PROGRAM PRG_ControlHMIInit
VAR
	(*	Konfiguracja HMIManager		*)
	fbDedaultHMIConfiguration		: FB_DefaultHMIConfiguration;
	fbHMIConfigure					: FB_HMIConfigure;
	
END_VAR

IF (NOT GVL_SystemVariable.bControlHMIInit) THEN
	GVL_SystemVariable.bControlHMIInit := TRUE;
		(*	Konfiguracjia systemu HMI	*)
	fbHMIConfigure.AddConfiguration (fbConfigure := fbDedaultHMIConfiguration);
	PRG_ControlHMI.fbHMIManager.AddModulConfigure (fbHMIConfigure := fbHMIConfigure);
	
END_IF

END_PROGRAM

(* stored: Version 1.1.0.1
   POU PRG_ControlHMIInit: Id {9feea808-f820-0e23-2d25-71153216f220}, SpecialFunc None *)
